(* Logix 5000 project; controller NorthLineDepalletizerPLC vendor 1 type 14 code 106 rev 33.11; software revision 33.00; part 2 of 4 *)
(* tags used below, declared in another part *)
   AcknowledgeCameraImage : ALIAS FOR YRC1000_Rbt_Ctlr:O.Data[4].5;
   ActiveUserFrame : DINT;   // Currently Active Pallet
   CameraAngle : REAL;
   CameraOffsetX : REAL;
   CameraOffsetY : REAL;
   CameraScore : REAL;
   ChangingJob : BOOL;
   CoilLocationFound : ALIAS FOR YRC1000_Rbt_Ctlr:O.Data[4].6;
   CompleteState : DINT;
   delay_2832_Edge_Camera : TIMER;
   delay_2832_Edge_SearchLocation : TIMER;
   delay_2832_Middle_Camera : TIMER;
   delay_2832_Middle_SearchLocation : TIMER;
   delay_2832_PickLocation : TIMER;
   delay_3041_Edge_Camera : TIMER;
   delay_3041_Edge_SearchLocation : TIMER;
   delay_3041_Middle_Camera : TIMER;
   delay_3041_Middle_SearchLocation : TIMER;
   delay_3041_PickLocation : TIMER;
   delay_PalletComplete : TIMER;
   err_CameraFailed : BOOL;
   ErrorState : DINT;
   FailedCaptures : DINT;   // Number of times the camera failed to find the coil
   FoundPattern : DINT;
   Gripper_HoldingPart : ALIAS FOR YRC1000_Rbt_Ctlr:O.Data[4].7;
   HorizontalLineFound : BOOL;
   i : DINT;
   JobResults : PatternResult[4];   // Organized results from the most recent camera image
   LeftEdgeFound : ALIAS FOR YRC1000_Rbt_Ctlr:O.Data[6].7;
   LeftPalletComplete : ALIAS FOR YRC1000_Rbt_Ctlr:O.Data[4].0;
   LoopsFound : BOOL;   // Used to determine if we are looking at the wrong end of a single-stack coil
   msg_Read_SearchLocation : MESSAGE;
   msg_Write_CoilLocation : MESSAGE;
   msg_Write_SearchLocation : MESSAGE;
   ons_Reset_3041Edge : BOOL;
   ons_Reset_3041Middle : BOOL;
   ons_Reset_CI_2832Edge : BOOL;
   ons_Reset_CI_2832Middle : BOOL;
   ons_Reset_CI_3041Edge : BOOL;
   ons_Reset_CI_3041Middle : BOOL;
   ons_StartJob3041 : BOOL;
   Read_SearchLocation : BOOL;
   RightEdgeFound : ALIAS FOR YRC1000_Rbt_Ctlr:O.Data[7].0;
   RightPalletComplete : ALIAS FOR YRC1000_Rbt_Ctlr:O.Data[4].1;
   RobotCameraRequest : ALIAS FOR YRC1000_Rbt_Ctlr:I.Data[9].4;
   run_2832_CE : BOOL;
   run_3041_CE : BOOL;
   RunPalletComplete : BOOL;
   SearchLocation : DINT;   // Index of what part of the pallet the camera is looking at
   SelectedJobID : DINT;
   state_CaptureImage : DINT;
   state_Job0017 : DINT;
   state_Job2832 : DINT;
   state_Job2832_Edge : DINT;
   state_Job2832_Middle : DINT;
   state_Job3041 : DINT;
   state_Job3041_Edge : DINT;
   state_Job3041_Middle : DINT;
   state_PalletComplete : DINT;
   timer_Job2832_CameraError : TIMER;
   timer_Job3041_CameraError : TIMER;
   VerticalLineFound : BOOL;
   Write_CoilLocation : BOOL;
   Write_SearchLocation : BOOL;
(* MainProgram, continued *)

ROUTINE Job2832_Edge   (* ladder *)
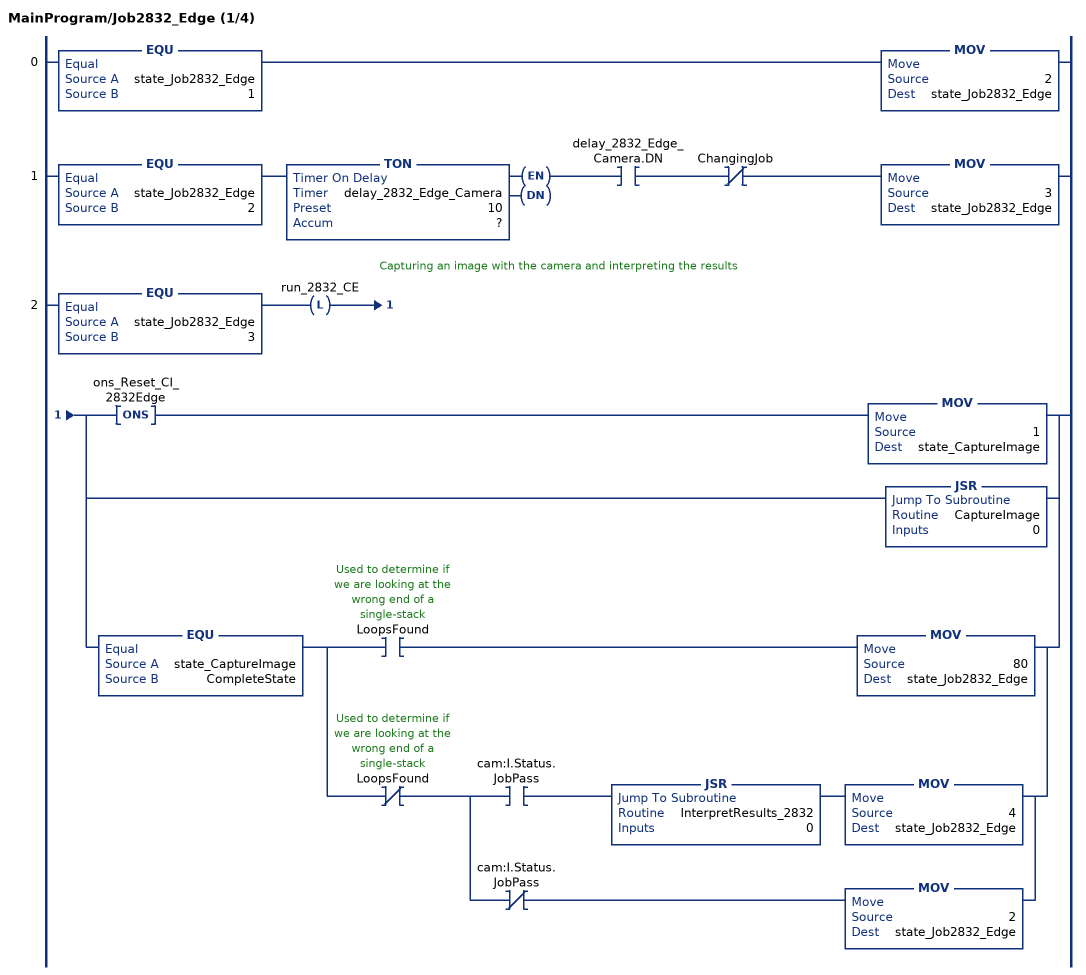
   0: EQU(state_Job2832_Edge,1)MOV(2,state_Job2832_Edge);
   1: EQU(state_Job2832_Edge,2)TON(delay_2832_Edge_Camera,?,?)XIC(delay_2832_Edge_Camera.DN)XIO(ChangingJob)MOV(3,state_Job2832_Edge);
   // Capturing an image with the camera and interpreting the results
   2: EQU(state_Job2832_Edge,3)OTL(run_2832_CE)[[ONS(ons_Reset_CI_2832Edge) MOV(1,state_CaptureImage) ,JSR(CaptureImage,0) ] ,EQU(state_CaptureImage,CompleteState) [XIC(LoopsFound) MOV(80,state_Job2832_Edge) ,XIO(LoopsFound) [XIC(cam:I.Status.JobPass) JSR(InterpretResults_2832,0) MOV(4,state_Job2832_Edge) ,XIO(cam:I.Status.JobPass) MOV(2,state_Job2832_Edge) ] ] ];
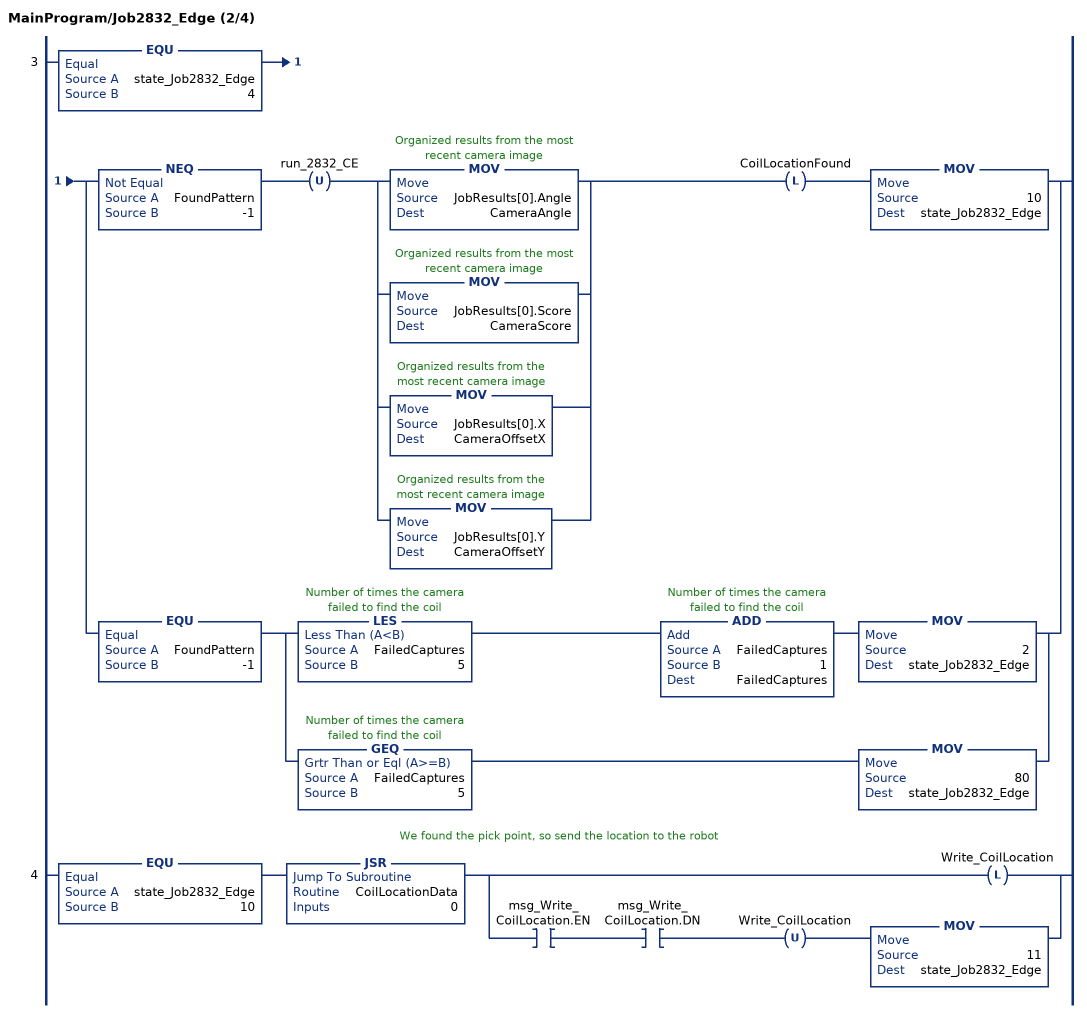
   3: EQU(state_Job2832_Edge,4)[NEQ(FoundPattern,-1) OTU(run_2832_CE) [MOV(JobResults[0].Angle,CameraAngle) ,MOV(JobResults[0].Score,CameraScore) ,MOV(JobResults[0].X,CameraOffsetX) ,MOV(JobResults[0].Y,CameraOffsetY) ] OTL(CoilLocationFound) MOV(10,state_Job2832_Edge) ,EQU(FoundPattern,-1) [LES(FailedCaptures,5) ADD(FailedCaptures,1,FailedCaptures) MOV(2,state_Job2832_Edge) ,GEQ(FailedCaptures,5) MOV(80,state_Job2832_Edge) ] ];
   // We found the pick point, so send the location to the robot
   4: EQU(state_Job2832_Edge,10)JSR(CoilLocationData,0)[OTL(Write_CoilLocation) ,XIC(msg_Write_CoilLocation.EN) XIC(msg_Write_CoilLocation.DN) OTU(Write_CoilLocation) MOV(11,state_Job2832_Edge) ];
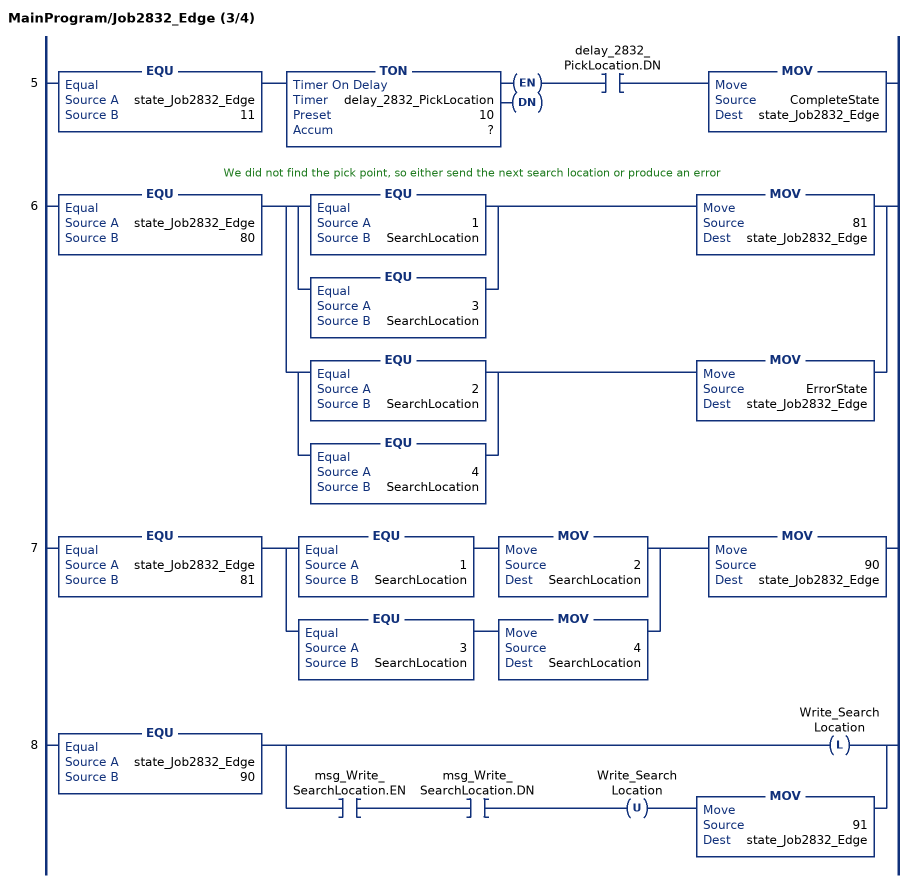
   5: EQU(state_Job2832_Edge,11)TON(delay_2832_PickLocation,?,?)XIC(delay_2832_PickLocation.DN)MOV(CompleteState,state_Job2832_Edge);
   // We did not find the pick point, so either send the next search location or produce an error
   6: EQU(state_Job2832_Edge,80)[[EQU(1,SearchLocation) ,EQU(3,SearchLocation) ] MOV(81,state_Job2832_Edge) ,[EQU(2,SearchLocation) ,EQU(4,SearchLocation) ] MOV(ErrorState,state_Job2832_Edge) ];
   7: EQU(state_Job2832_Edge,81)[EQU(1,SearchLocation) MOV(2,SearchLocation) ,EQU(3,SearchLocation) MOV(4,SearchLocation) ]MOV(90,state_Job2832_Edge);
   8: EQU(state_Job2832_Edge,90)[OTL(Write_SearchLocation) ,XIC(msg_Write_SearchLocation.EN) XIC(msg_Write_SearchLocation.DN) OTU(Write_SearchLocation) MOV(91,state_Job2832_Edge) ];
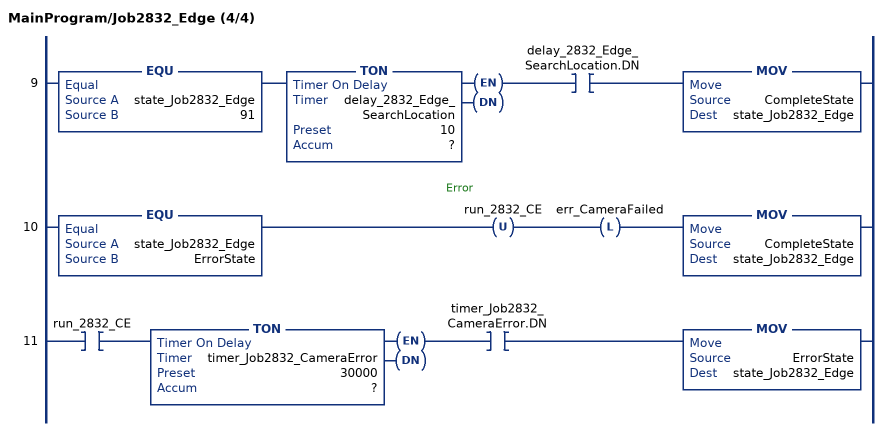
   9: EQU(state_Job2832_Edge,91)TON(delay_2832_Edge_SearchLocation,?,?)XIC(delay_2832_Edge_SearchLocation.DN)MOV(CompleteState,state_Job2832_Edge);
   // Error
   10: EQU(state_Job2832_Edge,ErrorState)OTU(run_2832_CE)OTL(err_CameraFailed)MOV(CompleteState,state_Job2832_Edge);
   11: XIC(run_2832_CE)TON(timer_Job2832_CameraError,?,?)XIC(timer_Job2832_CameraError.DN)MOV(ErrorState,state_Job2832_Edge);
END_ROUTINE

ROUTINE Job2832_Middle   (* ladder *)
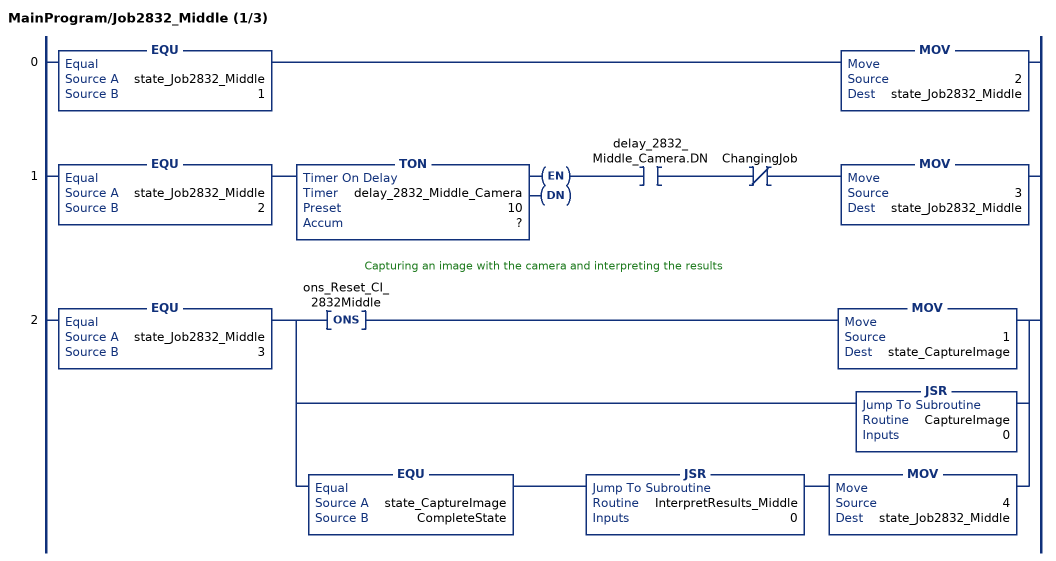
   0: EQU(state_Job2832_Middle,1)MOV(2,state_Job2832_Middle);
   1: EQU(state_Job2832_Middle,2)TON(delay_2832_Middle_Camera,?,?)XIC(delay_2832_Middle_Camera.DN)XIO(ChangingJob)MOV(3,state_Job2832_Middle);
   // Capturing an image with the camera and interpreting the results
   2: EQU(state_Job2832_Middle,3)[[ONS(ons_Reset_CI_2832Middle) MOV(1,state_CaptureImage) ,JSR(CaptureImage,0) ] ,EQU(state_CaptureImage,CompleteState) JSR(InterpretResults_Middle,0) MOV(4,state_Job2832_Middle) ];
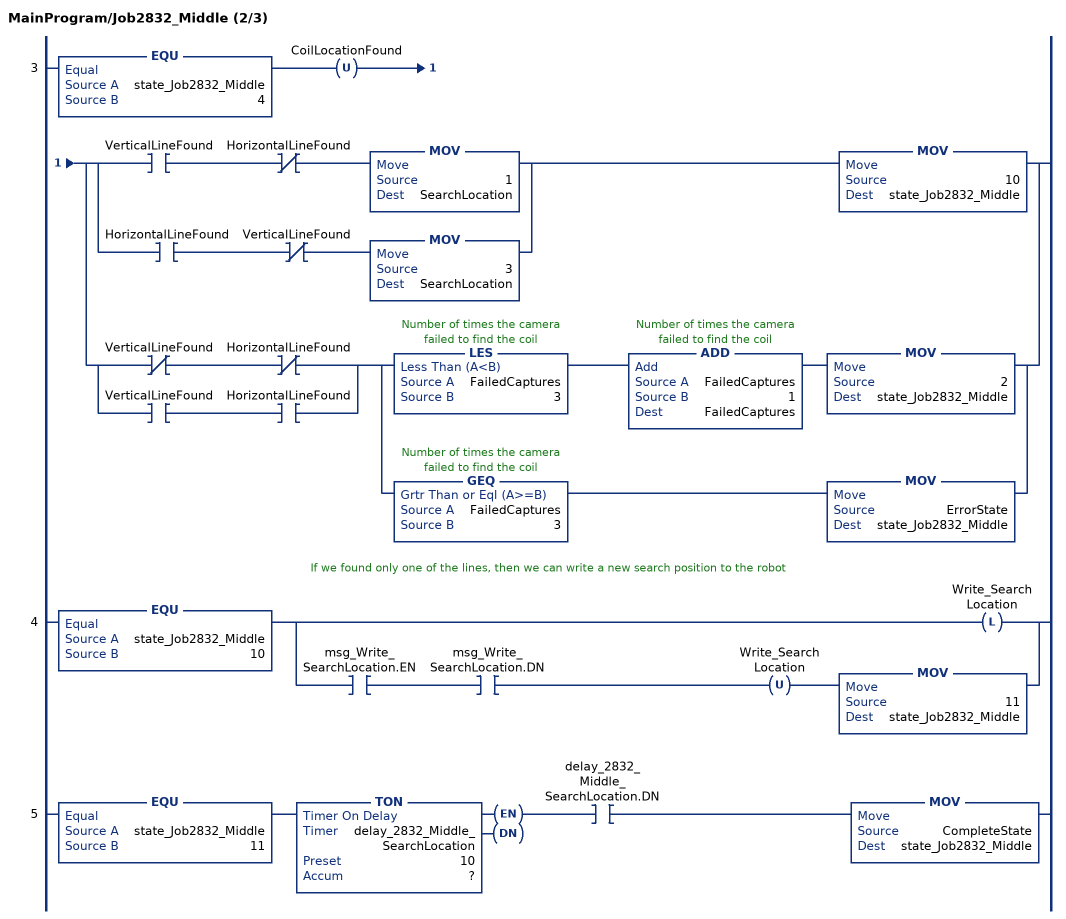
   3: EQU(state_Job2832_Middle,4)OTU(CoilLocationFound)[[XIC(VerticalLineFound) XIO(HorizontalLineFound) MOV(1,SearchLocation) ,XIC(HorizontalLineFound) XIO(VerticalLineFound) MOV(3,SearchLocation) ] MOV(10,state_Job2832_Middle) ,[XIO(VerticalLineFound) XIO(HorizontalLineFound) ,XIC(VerticalLineFound) XIC(HorizontalLineFound) ] [LES(FailedCaptures,3) ADD(FailedCaptures,1,FailedCaptures) MOV(2,state_Job2832_Middle) ,GEQ(FailedCaptures,3) MOV(ErrorState,state_Job2832_Middle) ] ];
   // If we found only one of the lines, then we can write a new search position to the robot
   4: EQU(state_Job2832_Middle,10)[OTL(Write_SearchLocation) ,XIC(msg_Write_SearchLocation.EN) XIC(msg_Write_SearchLocation.DN) OTU(Write_SearchLocation) MOV(11,state_Job2832_Middle) ];
   5: EQU(state_Job2832_Middle,11)TON(delay_2832_Middle_SearchLocation,?,?)XIC(delay_2832_Middle_SearchLocation.DN)MOV(CompleteState,state_Job2832_Middle);
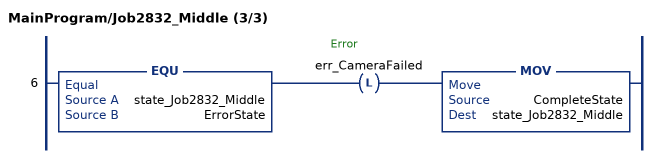
   // Error
   6: EQU(state_Job2832_Middle,ErrorState)OTL(err_CameraFailed)MOV(CompleteState,state_Job2832_Middle);
END_ROUTINE

ROUTINE Job3041   (* ladder *)
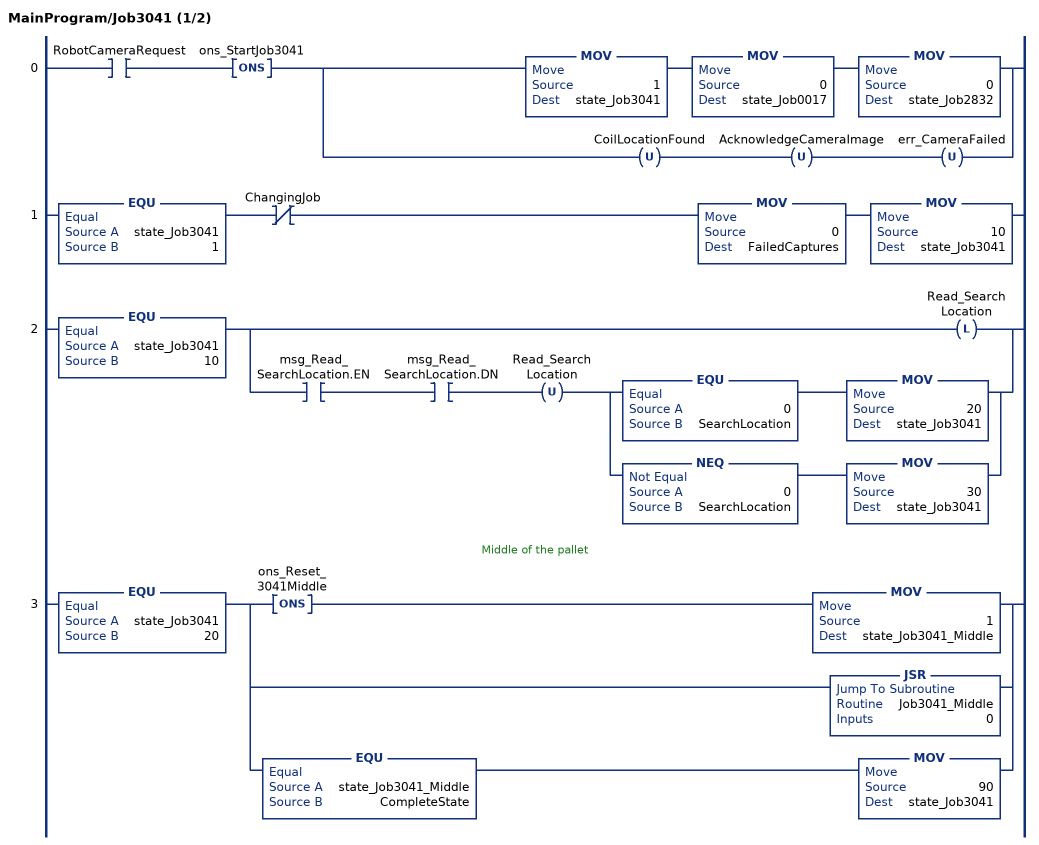
   0: XIC(RobotCameraRequest)ONS(ons_StartJob3041)[MOV(1,state_Job3041) MOV(0,state_Job0017) MOV(0,state_Job2832) ,OTU(CoilLocationFound) OTU(AcknowledgeCameraImage) OTU(err_CameraFailed) ];
   1: EQU(state_Job3041,1)XIO(ChangingJob)MOV(0,FailedCaptures)MOV(10,state_Job3041);
   2: EQU(state_Job3041,10)[OTL(Read_SearchLocation) ,XIC(msg_Read_SearchLocation.EN) XIC(msg_Read_SearchLocation.DN) OTU(Read_SearchLocation) [EQU(0,SearchLocation) MOV(20,state_Job3041) ,NEQ(0,SearchLocation) MOV(30,state_Job3041) ] ];
   // Middle of the pallet
   3: EQU(state_Job3041,20)[[ONS(ons_Reset_3041Middle) MOV(1,state_Job3041_Middle) ,JSR(Job3041_Middle,0) ] ,EQU(state_Job3041_Middle,CompleteState) MOV(90,state_Job3041) ];
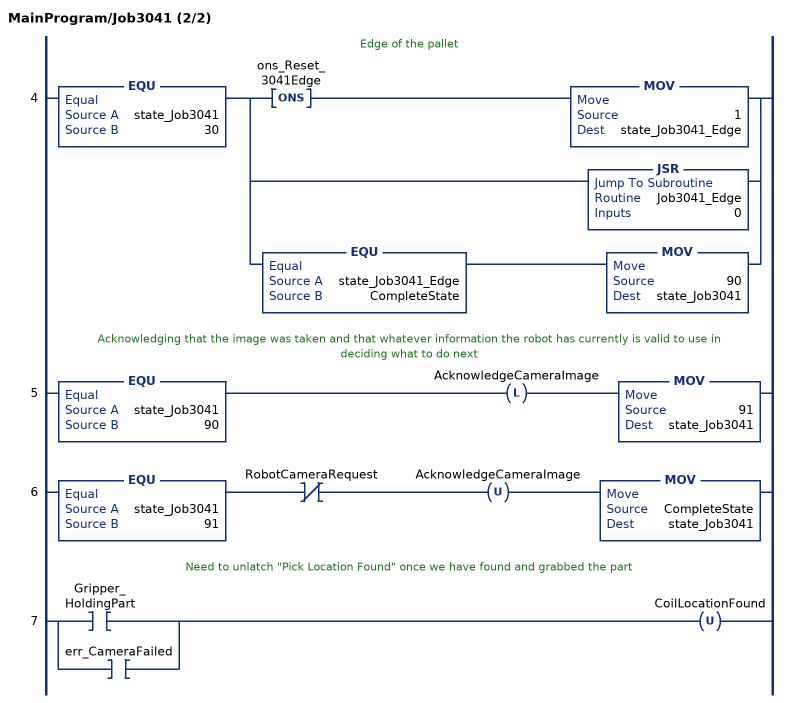
   // Edge of the pallet
   4: EQU(state_Job3041,30)[[ONS(ons_Reset_3041Edge) MOV(1,state_Job3041_Edge) ,JSR(Job3041_Edge,0) ] ,EQU(state_Job3041_Edge,CompleteState) MOV(90,state_Job3041) ];
   // Acknowledging that the image was taken and that whatever information the robot has currently is valid to use in deciding what to do next
   5: EQU(state_Job3041,90)OTL(AcknowledgeCameraImage)MOV(91,state_Job3041);
   6: EQU(state_Job3041,91)XIO(RobotCameraRequest)OTU(AcknowledgeCameraImage)MOV(CompleteState,state_Job3041);
   // Need to unlatch "Pick Location Found" once we have found and grabbed the part
   7: [XIC(Gripper_HoldingPart) ,XIC(err_CameraFailed) ]OTU(CoilLocationFound);
END_ROUTINE

ROUTINE Job3041_Edge   (* ladder *)
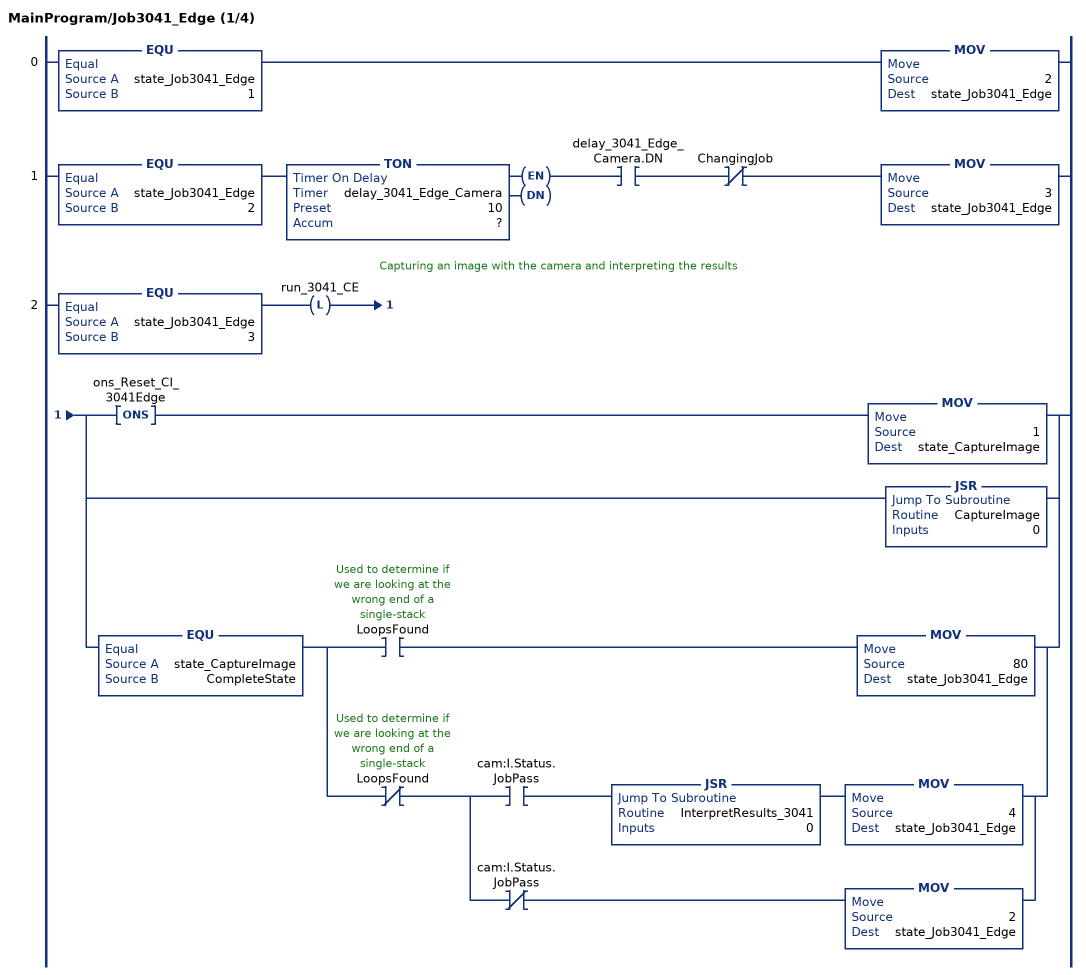
   0: EQU(state_Job3041_Edge,1)MOV(2,state_Job3041_Edge);
   1: EQU(state_Job3041_Edge,2)TON(delay_3041_Edge_Camera,?,?)XIC(delay_3041_Edge_Camera.DN)XIO(ChangingJob)MOV(3,state_Job3041_Edge);
   // Capturing an image with the camera and interpreting the results
   2: EQU(state_Job3041_Edge,3)OTL(run_3041_CE)[[ONS(ons_Reset_CI_3041Edge) MOV(1,state_CaptureImage) ,JSR(CaptureImage,0) ] ,EQU(state_CaptureImage,CompleteState) [XIC(LoopsFound) MOV(80,state_Job3041_Edge) ,XIO(LoopsFound) [XIC(cam:I.Status.JobPass) JSR(InterpretResults_3041,0) MOV(4,state_Job3041_Edge) ,XIO(cam:I.Status.JobPass) MOV(2,state_Job3041_Edge) ] ] ];
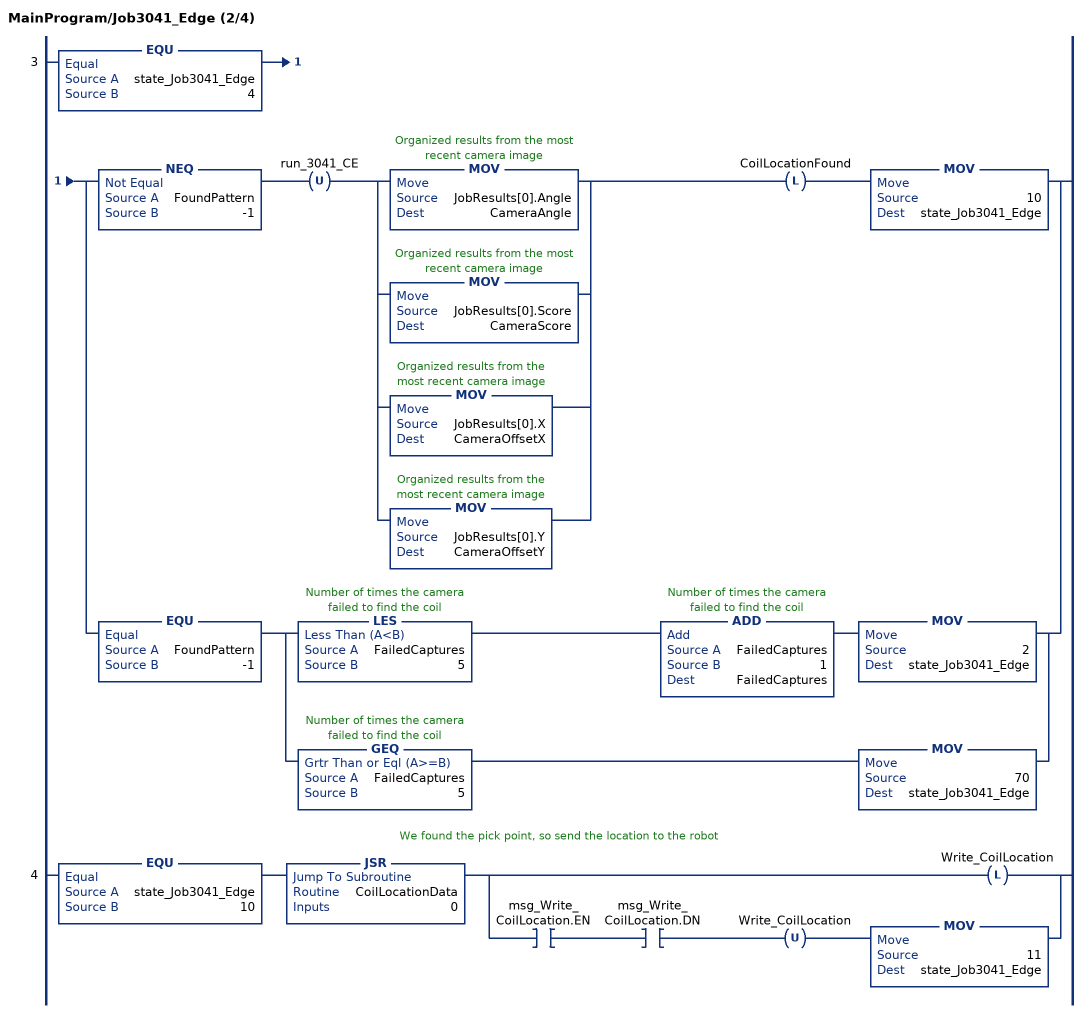
   3: EQU(state_Job3041_Edge,4)[NEQ(FoundPattern,-1) OTU(run_3041_CE) [MOV(JobResults[0].Angle,CameraAngle) ,MOV(JobResults[0].Score,CameraScore) ,MOV(JobResults[0].X,CameraOffsetX) ,MOV(JobResults[0].Y,CameraOffsetY) ] OTL(CoilLocationFound) MOV(10,state_Job3041_Edge) ,EQU(FoundPattern,-1) [LES(FailedCaptures,5) ADD(FailedCaptures,1,FailedCaptures) MOV(2,state_Job3041_Edge) ,GEQ(FailedCaptures,5) MOV(70,state_Job3041_Edge) ] ];
   // We found the pick point, so send the location to the robot
   4: EQU(state_Job3041_Edge,10)JSR(CoilLocationData,0)[OTL(Write_CoilLocation) ,XIC(msg_Write_CoilLocation.EN) XIC(msg_Write_CoilLocation.DN) OTU(Write_CoilLocation) MOV(11,state_Job3041_Edge) ];
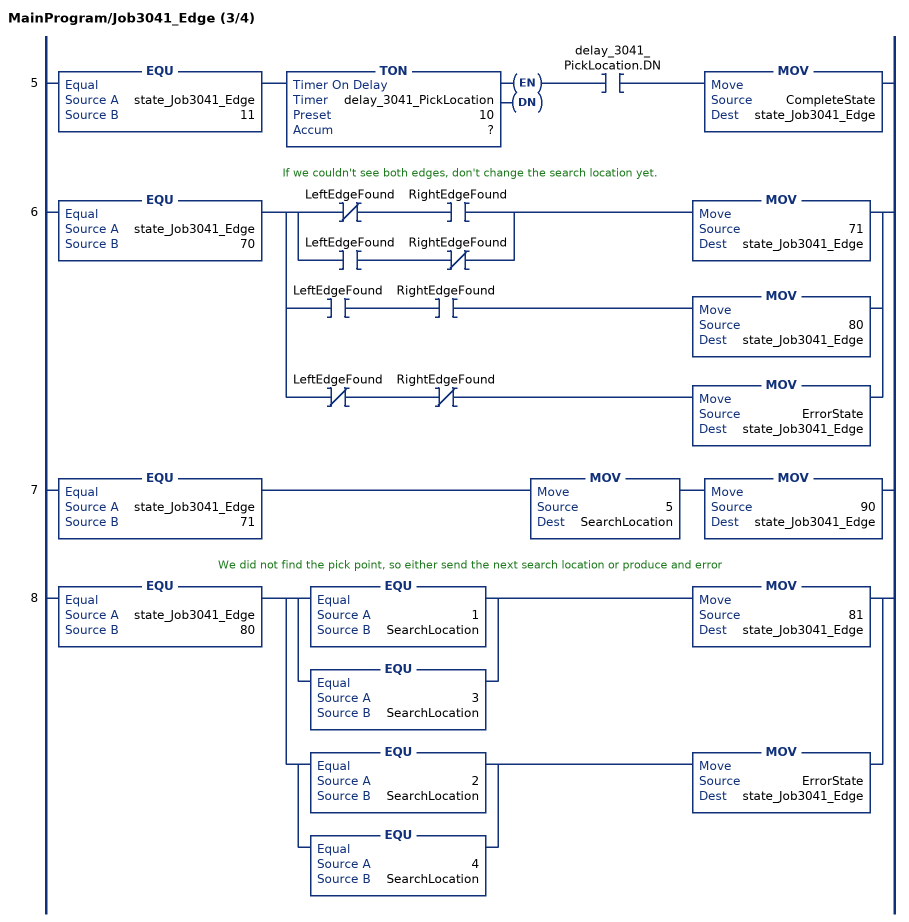
   5: EQU(state_Job3041_Edge,11)TON(delay_3041_PickLocation,?,?)XIC(delay_3041_PickLocation.DN)MOV(CompleteState,state_Job3041_Edge);
   // If we couldn't see both edges, don't change the search location yet.
   6: EQU(state_Job3041_Edge,70)[[XIO(LeftEdgeFound) XIC(RightEdgeFound) ,XIC(LeftEdgeFound) XIO(RightEdgeFound) ] MOV(71,state_Job3041_Edge) ,XIC(LeftEdgeFound) XIC(RightEdgeFound) MOV(80,state_Job3041_Edge) ,XIO(LeftEdgeFound) XIO(RightEdgeFound) MOV(ErrorState,state_Job3041_Edge) ];
   7: EQU(state_Job3041_Edge,71)MOV(5,SearchLocation)MOV(90,state_Job3041_Edge);
   // We did not find the pick point, so either send the next search location or produce and error
   8: EQU(state_Job3041_Edge,80)[[EQU(1,SearchLocation) ,EQU(3,SearchLocation) ] MOV(81,state_Job3041_Edge) ,[EQU(2,SearchLocation) ,EQU(4,SearchLocation) ] MOV(ErrorState,state_Job3041_Edge) ];
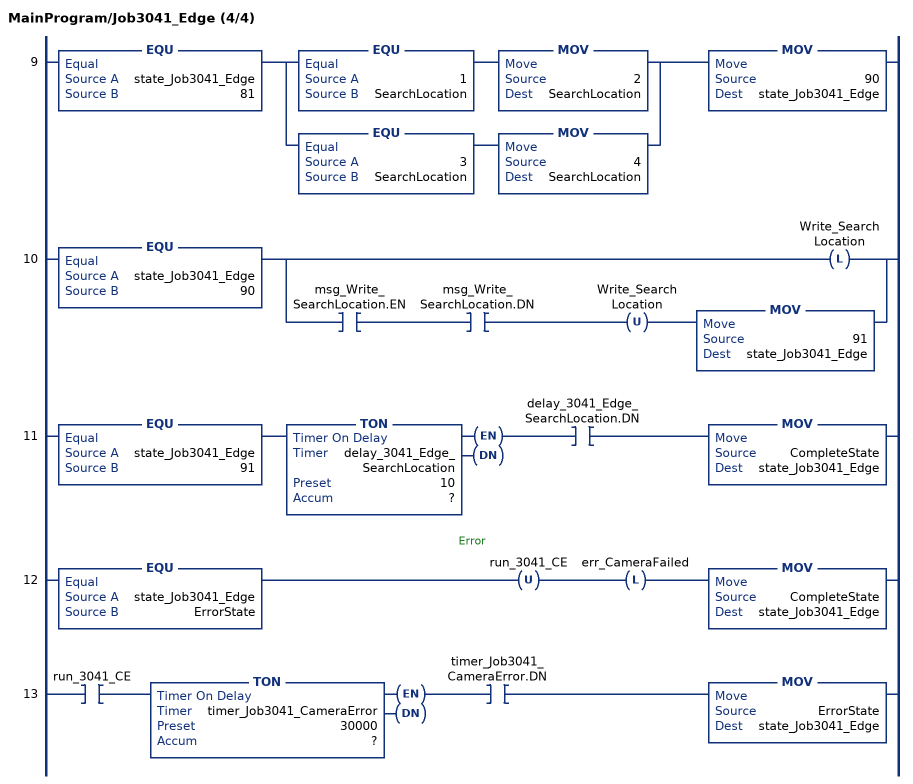
   9: EQU(state_Job3041_Edge,81)[EQU(1,SearchLocation) MOV(2,SearchLocation) ,EQU(3,SearchLocation) MOV(4,SearchLocation) ]MOV(90,state_Job3041_Edge);
   10: EQU(state_Job3041_Edge,90)[OTL(Write_SearchLocation) ,XIC(msg_Write_SearchLocation.EN) XIC(msg_Write_SearchLocation.DN) OTU(Write_SearchLocation) MOV(91,state_Job3041_Edge) ];
   11: EQU(state_Job3041_Edge,91)TON(delay_3041_Edge_SearchLocation,?,?)XIC(delay_3041_Edge_SearchLocation.DN)MOV(CompleteState,state_Job3041_Edge);
   // Error
   12: EQU(state_Job3041_Edge,ErrorState)OTU(run_3041_CE)OTL(err_CameraFailed)MOV(CompleteState,state_Job3041_Edge);
   13: XIC(run_3041_CE)TON(timer_Job3041_CameraError,?,?)XIC(timer_Job3041_CameraError.DN)MOV(ErrorState,state_Job3041_Edge);
END_ROUTINE

ROUTINE Job3041_Middle   (* ladder *)
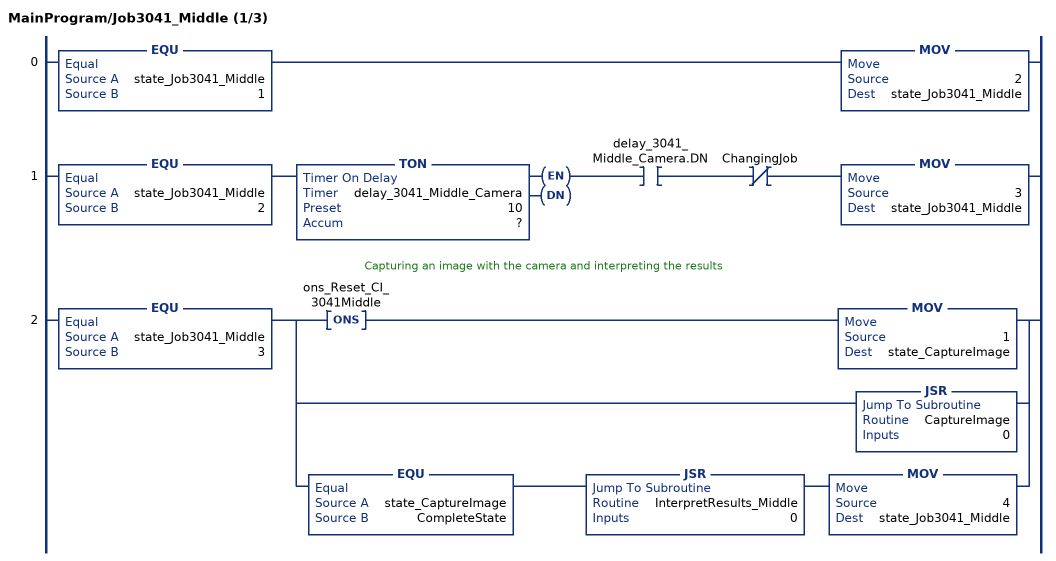
   0: EQU(state_Job3041_Middle,1)MOV(2,state_Job3041_Middle);
   1: EQU(state_Job3041_Middle,2)TON(delay_3041_Middle_Camera,?,?)XIC(delay_3041_Middle_Camera.DN)XIO(ChangingJob)MOV(3,state_Job3041_Middle);
   // Capturing an image with the camera and interpreting the results
   2: EQU(state_Job3041_Middle,3)[[ONS(ons_Reset_CI_3041Middle) MOV(1,state_CaptureImage) ,JSR(CaptureImage,0) ] ,EQU(state_CaptureImage,CompleteState) JSR(InterpretResults_Middle,0) MOV(4,state_Job3041_Middle) ];
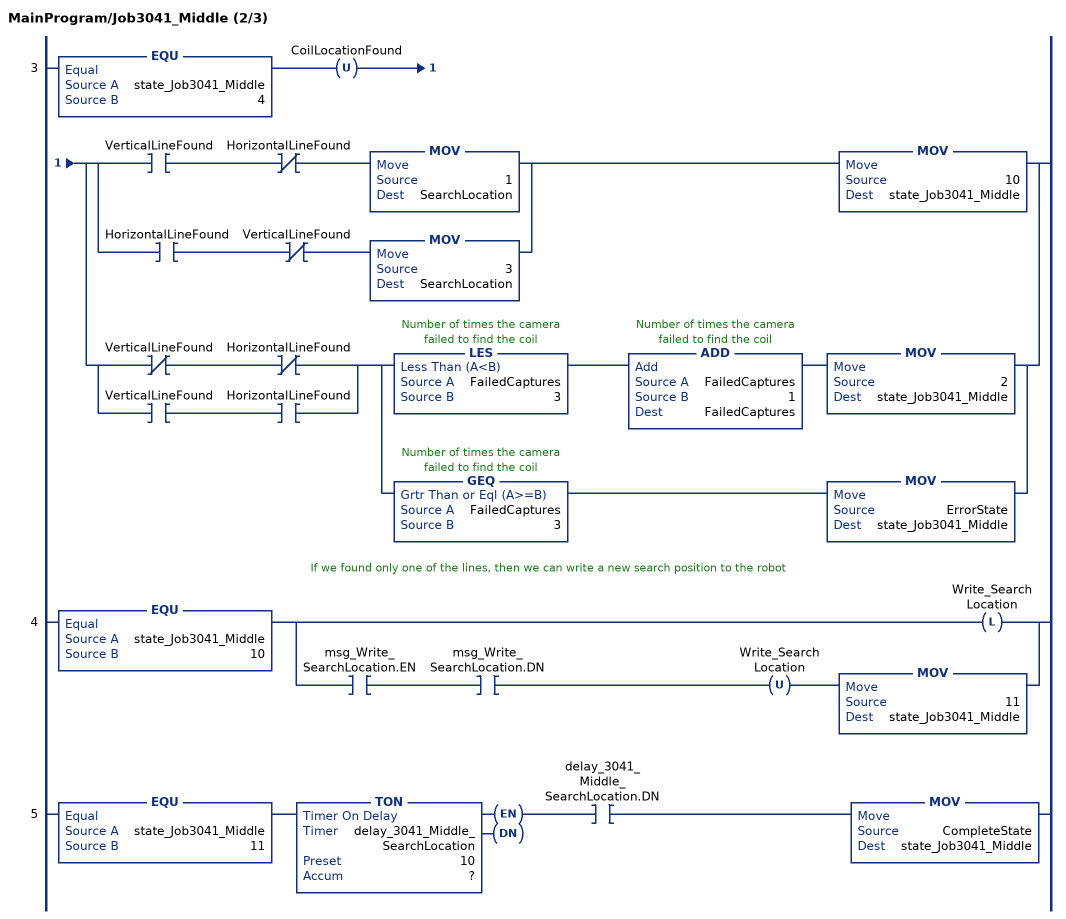
   3: EQU(state_Job3041_Middle,4)OTU(CoilLocationFound)[[XIC(VerticalLineFound) XIO(HorizontalLineFound) MOV(1,SearchLocation) ,XIC(HorizontalLineFound) XIO(VerticalLineFound) MOV(3,SearchLocation) ] MOV(10,state_Job3041_Middle) ,[XIO(VerticalLineFound) XIO(HorizontalLineFound) ,XIC(VerticalLineFound) XIC(HorizontalLineFound) ] [LES(FailedCaptures,3) ADD(FailedCaptures,1,FailedCaptures) MOV(2,state_Job3041_Middle) ,GEQ(FailedCaptures,3) MOV(ErrorState,state_Job3041_Middle) ] ];
   // If we found only one of the lines, then we can write a new search position to the robot
   4: EQU(state_Job3041_Middle,10)[OTL(Write_SearchLocation) ,XIC(msg_Write_SearchLocation.EN) XIC(msg_Write_SearchLocation.DN) OTU(Write_SearchLocation) MOV(11,state_Job3041_Middle) ];
   5: EQU(state_Job3041_Middle,11)TON(delay_3041_Middle_SearchLocation,?,?)XIC(delay_3041_Middle_SearchLocation.DN)MOV(CompleteState,state_Job3041_Middle);
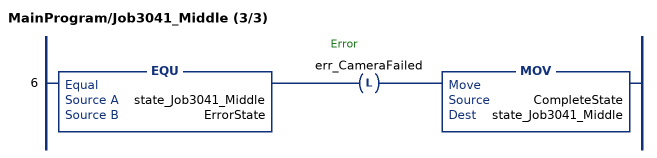
   // Error
   6: EQU(state_Job3041_Middle,ErrorState)OTL(err_CameraFailed)MOV(CompleteState,state_Job3041_Middle);
END_ROUTINE

ROUTINE Main   (* ladder *)
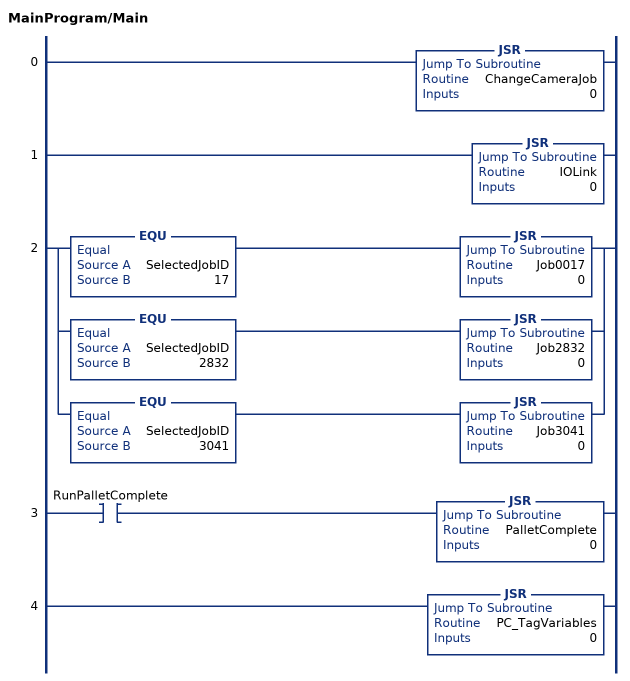
   0: JSR(ChangeCameraJob,0);
   1: JSR(IOLink,0);
   2: [EQU(SelectedJobID,17) JSR(Job0017,0) ,EQU(SelectedJobID,2832) JSR(Job2832,0) ,EQU(SelectedJobID,3041) JSR(Job3041,0) ];
   3: XIC(RunPalletComplete)JSR(PalletComplete,0);
   4: JSR(PC_TagVariables,0);
END_ROUTINE

ROUTINE PalletComplete   (* ladder *)
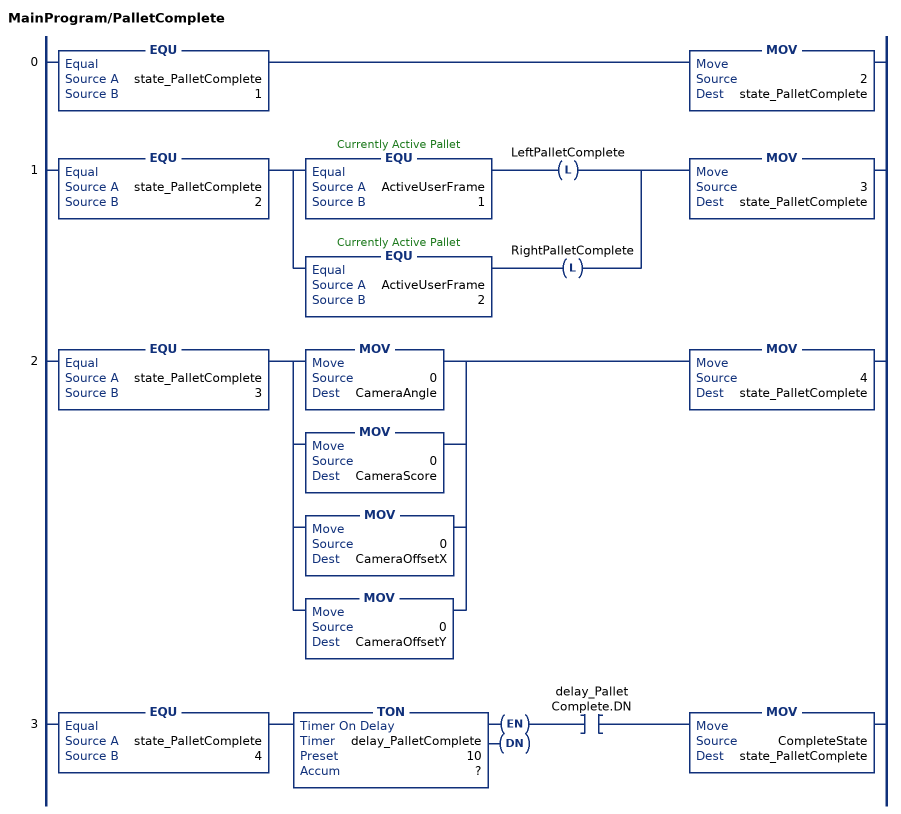
   0: EQU(state_PalletComplete,1)MOV(2,state_PalletComplete);
   1: EQU(state_PalletComplete,2)[EQU(ActiveUserFrame,1) OTL(LeftPalletComplete) ,EQU(ActiveUserFrame,2) OTL(RightPalletComplete) ]MOV(3,state_PalletComplete);
   2: EQU(state_PalletComplete,3)[MOV(0,CameraAngle) ,MOV(0,CameraScore) ,MOV(0,CameraOffsetX) ,MOV(0,CameraOffsetY) ]MOV(4,state_PalletComplete);
   3: EQU(state_PalletComplete,4)TON(delay_PalletComplete,?,?)XIC(delay_PalletComplete.DN)MOV(CompleteState,state_PalletComplete);
END_ROUTINE
